FUNCTION_BLOCK ABSTRACT GenericSubarea
VAR_IN_OUT
	bundlesQueue : ARRAY[*] OF Bundle;
	bundlesBypass : ARRAY[*] OF BOOL;
	
	//ecDevices : ARRAY[0..EC_MAX_SLAVES] OF ST_EcSlaveConfigData; //devices
	ecDeviceStates : ARRAY[*] OF ST_EcSlaveState; //device states
END_VAR
VAR_INPUT
	ecIndex0, ecIndex1 : DINT;
END_VAR
VAR_OUTPUT //controls
	stop AT %I* : BOOL;
	
	ready : BOOL;
	active : BOOL;
	error : BOOL;
	
	ecNetworkError : BOOL;
END_VAR

CheckEcNetwork(
	ecDeviceStates:= ecDeviceStates, 
	ecIndex0:= ecIndex0, 
	ecIndex1:= ecIndex1, 
	errorInit=> , 
	errorPreop=> , 
	errorBootstrap=> , 
	errorSafeop=> , 
	error=> ecNetworkError, 
	operational=> );
	
callHardware();

setupHardware();

runModules();

callHardware();

METHOD PROTECTED ABSTRACT callHardware : BOOL
VAR_INPUT
END_VAR
END_METHOD

METHOD PROTECTED ABSTRACT runModules : BOOL
VAR_INPUT
END_VAR
END_METHOD

METHOD PROTECTED ABSTRACT setupHardware : BOOL
VAR_INPUT
END_VAR
END_METHOD

END_FUNCTION_BLOCK

(* stored: Version 1.1.0.1, ProductVersion 3.1.4024.11
   POU GenericSubarea: Id {b8afc32a-0b49-49f1-91d4-4409bf7ce05b}, SpecialFunc None
   Folder Abstract: Id {025764d4-c739-47cc-a99c-055f76ffc6c8}
   Method callHardware: Id {842b4e14-ad00-4a54-ad2e-783f2d1be972}
   Method runModules: Id {7a7ff579-c078-4df6-bea2-4df6e9ceeed4}
   Method setupHardware: Id {632a9403-7ef3-48d3-bc64-595606118f92} *)
